// TwinCAT 3 PLC project Fraktal_Demo
// Title: Fraktal_Demo
// Company: fraktal-automation
// Author: fraktal-automation
// ProjectVersion: 0.1.0.4
// Description: Executable two-root Fraktal demonstration application. Not a reusable library.
// ProgramVersion: 3.1.4024.0
// libraries:
//   Tc2_Standard, * (Beckhoff Automation GmbH)
//   Tc3_Module, * (Beckhoff Automation GmbH)
//   Fraktal_Core, 0.25.0.0 (fraktal-automation)
//   Fraktal_Modules, 0.11.0.3 (fraktal-automation)
// project tree:
//   / PlcTask.TcTTO (not stored)
//   00_System/ MAIN.TcPOU
//   01_ClampCell/ FB_ClampCellUnit.TcPOU
//   01_ClampCell/Sequences/ FB_ClampCellAuto.TcPOU
// real-time tasks:
//   TASK PlcTask: cycle T#10ms, priority 20, ADS port 350

// ---- 00_System/MAIN.TcPOU
// Core §4.2 — a program with a FOREST of root Units (two independent stations).
// Each root is ticked every scan; each owns its mode, cycle, model, and rollup.
// The HMI (§3.13) may show both roots or scope to one.
PROGRAM MAIN
VAR
    Recipe  : FB_LocalRecipeProvider;
    // --- two peer roots (no shared super-root in PLC code) ---
    {attribute 'OPC.UA.DA' := '1'}
    ClampCellA : FB_ClampCellUnit;
    {attribute 'OPC.UA.DA' := '1'}
    ClampCellB : FB_ClampCellUnit;
    _init : BOOL;
    _plate : ST_Nameplate;   // §3.10.1 example identity
    _modelA, _modelB : ST_ModelId;
    HalA1, HalA2, HalB1, HalB2 : ST_CylinderHal;
    SimA1, SimA2, SimB1, SimB2 : FB_CylinderSim;
    CylPar : ST_CylinderParCfg;
    ClampPar : ST_ClampParCfg;
END_VAR

IF NOT _init THEN
    _init := TRUE;
    Recipe.Register(ModelCode := '', RecipeKey := 'CylinderCM', pData := ADR(CylPar), Size := SIZEOF(CylPar));
    Recipe.Register(ModelCode := '', RecipeKey := 'ClampEM',    pData := ADR(ClampPar), Size := SIZEOF(ClampPar));
    ClampCellA.Setup(Name := 'ClampCellA', HalA := HalA1, HalB := HalA2, Recipe := Recipe);
    ClampCellB.Setup(Name := 'ClampCellB', HalA := HalB1, HalB := HalB2, Recipe := Recipe);
    SimA1.Setup(HalRef := HalA1, TravelTime := T#0S);
    SimA2.Setup(HalRef := HalA2, TravelTime := T#0S);
    SimB1.Setup(HalRef := HalB1, TravelTime := T#0S);
    SimB2.Setup(HalRef := HalB2, TravelTime := T#0S);
    _modelA.ModelCode := 'CLAMP-A';
    _modelB.ModelCode := 'CLAMP-B';
    ClampCellA.SetModel(Id := _modelA);
    ClampCellB.SetModel(Id := _modelB);
    // §3.10.1: a root Unit SHALL publish a digital nameplate (identity set at the
    // instantiation site — the machine builder knows what was shipped, not the type)
    _plate.ProductUri         := 'https://example.org/assets/clampcell/SN-2026-0001';
    _plate.ManufacturerName   := 'Example Machines GmbH';
    _plate.ProductDesignation := 'Dual-Cylinder Clamp Cell';
    _plate.SerialNumber       := 'SN-2026-0001';
    _plate.YearOfConstruction := '2026';
    _plate.SoftwareVersion    := 'Fraktal 1.0';
    _plate.DocumentationUrl   := 'https://example.org/docs/clampcell';
    ClampCellA.SetNameplate(Plate := _plate);
    // §8.9 standard reason metadata is generated and manifest-served by the Unit.
    _plate.SerialNumber       := 'SN-2026-0002';
    _plate.ProductUri         := 'https://example.org/assets/clampcell/SN-2026-0002';
    ClampCellB.SetNameplate(Plate := _plate);
END_IF
// simulated plant, then the two independent roots:
SimA1();
SimA2();
SimB1();
SimB2();
ClampCellA();
ClampCellB();

END_PROGRAM

// ---- 01_ClampCell/FB_ClampCellUnit.TcPOU
// Project-owned root Unit of the core demo: one clamp EM from the reusable library,
// cycled clamp -> unclamp by the AUTO chain. Wiring only (§6.8): every step lives
// in FB_ClampCellAuto, and the base restarts that chain on first scan, mode change
// and abort, so this type writes no lifecycle glue (§1.1 O1).
FUNCTION_BLOCK FB_ClampCellUnit EXTENDS FB_UnitBase
VAR_OUTPUT
    Clamp : FB_ClampEM;
END_VAR
VAR
    {attribute 'OPC.UA.DA' := '0'}
    _autoSequence : FB_ClampCellAuto;
END_VAR

Cyclic();

METHOD Setup : BOOL
VAR_INPUT
    Name : STRING(80);
    HalA : REFERENCE TO ST_CylinderHal;
    HalB : REFERENCE TO ST_CylinderHal;
    Recipe : I_RecipeProvider;
END_VAR
_M_SetName(Name);
_M_SetPresentation(DisplayNameKey := 'project.module.clampCell.name',
    DescriptionKey := 'project.module.clampCell.description',
    TypeKey := 'project.moduleType.clampCell');
Setup := Clamp.Setup(Name := CONCAT(Name, '.Clamp'), HalA := HalA, HalB := HalB, Recipe := Recipe)
    AND _M_Register(Child := Clamp)
    AND _autoSequence.Setup(Host := THIS^, Clamp := Clamp);
END_METHOD

// Thin mode router: AUTO runs the chain; MANUAL commands the clamp directly.
METHOD PROTECTED _M_Dispatch
CASE ModeActive OF
    E_Mode.AUTO:
        _autoSequence.M_Run();
ELSE
    _M_Fault(E_Reason.UNSUPPORTED_COMMAND, 'project.error.clampCellModeHasNoSequence');
END_CASE
END_METHOD

END_FUNCTION_BLOCK

// ---- 01_ClampCell/Sequences/FB_ClampCellAuto.TcPOU
// §6.8 AUTO chain of the clamp cell: clamp, unclamp, loop. Each command step names
// the clamp in Awaits, so a stall or a child fault is explained by the base walk
// (§6.9) - the chain writes no diagnostic of its own.
FUNCTION_BLOCK FB_ClampCellAuto EXTENDS FB_SequenceBase
VAR
    {attribute 'OPC.UA.DA' := '0'}
    _clamp : REFERENCE TO FB_ClampEM;
END_VAR

;

METHOD Setup : BOOL
VAR_INPUT
    Host : I_SequenceHost;
END_VAR
VAR_IN_OUT
    Clamp : FB_ClampEM;
END_VAR
_clamp REF= Clamp;
Setup := M_Attach(Host := Host) AND __ISVALIDREF(_clamp);
END_METHOD

METHOD M_Run
CASE _step OF
    0:
        M_Step(StepNo := 0, StepName := 'project.step.clampCellStart',
            Awaits := 0, AwaitingLabel := '', TimeClass := E_TimeClass.WORK, ExpectedTime := T#0S, Branch := 0);
        _retVal := E_StepResult.ADVANCE;
        M_Advance(OnAdvance := 100, OnJump1 := -1, OnJump2 := -1, OnJump3 := -1);
    100:
        M_Step(StepNo := 100, StepName := 'project.step.clampCellClamp',
            Awaits := _clamp, AwaitingLabel := 'Clamp.CLAMP', TimeClass := E_TimeClass.WORK, ExpectedTime := T#0S, Branch := 0);
        IF M_TryIssue(Steppable := TRUE) THEN
            _clamp.Abort := FALSE; _clamp.Command := E_ClampCommand.CLAMP; _clamp.Execute := TRUE;
        END_IF
        IF _clamp.Done THEN
            _clamp.Execute := FALSE;
            _retVal := E_StepResult.ADVANCE;
        END_IF
        M_Advance(OnAdvance := 200, OnJump1 := -1, OnJump2 := -1, OnJump3 := -1);
    200:
        M_Step(StepNo := 200, StepName := 'project.step.clampCellUnclamp',
            Awaits := _clamp, AwaitingLabel := 'Clamp.UNCLAMP', TimeClass := E_TimeClass.WORK, ExpectedTime := T#0S, Branch := 0);
        IF M_TryIssue(Steppable := TRUE) THEN
            _clamp.Abort := FALSE; _clamp.Command := E_ClampCommand.UNCLAMP; _clamp.Execute := TRUE;
        END_IF
        IF _clamp.Done THEN
            _clamp.Execute := FALSE;
            _retVal := E_StepResult.ADVANCE;
        END_IF
        M_Advance(OnAdvance := 999, OnJump1 := -1, OnJump2 := -1, OnJump3 := -1);
    999:  // cycle complete (§8.11.1 finish marker); loop unless a stop is pending
        M_Step(StepNo := 999, StepName := 'project.step.clampCellComplete',
            Awaits := 0, AwaitingLabel := '', TimeClass := E_TimeClass.WORK, ExpectedTime := T#0S, Branch := 0);
        IF M_EndOfCycle() THEN
            _retVal := E_StepResult.ADVANCE;
        END_IF
        M_Advance(OnAdvance := 100, OnJump1 := -1, OnJump2 := -1, OnJump3 := -1);
ELSE
    M_Fault(Reason := E_Reason.STEP_STALLED, DescriptionKey := 'std.error.undefinedStep');
END_CASE
END_METHOD

END_FUNCTION_BLOCK
